// TIA Portal V21 export
FUNCTION "GestPid_Comando1Motore" : Void   // FC62, LAD
{ S7_Optimized_Access := 'TRUE' }
// stored: SetENOAutomatically false
   VAR_INPUT
      K_Motore : Int;
      K_Pid : Int;
   END_VAR
BEGIN

REGION Network 1 (SCL)
   "Pid".P[#K_Pid].In.K_Motore1 := #K_Motore;
END_REGION
END_FUNCTION
